INTERFACE IEcTask EXTENDS ITask

PROPERTY NetID : amsnetid
GET
END_GET
SET
END_SET
END_PROPERTY

END_INTERFACE

(* stored: Version 1.1.0.1, ProductVersion 3.1.4024.9
   Itf IEcTask: Id {8a32a453-5ec2-43ef-95c2-50c158a5030e}
   Property NetID: Id {d5c28203-1370-4b4e-8cb8-15c09c3c79e0}
   Get Get: Id {5a077870-fc17-447c-a981-288a63c271f3}
   Set Set: Id {12a1e465-2387-462d-8ba1-d9b77af2ca45} *)
